Fanuc KAREL source: compact_preamble.KL

PROGRAM KD00043
%NOLOCKGROUP
VAR
I:INTEGER;J:INTEGER;B:BOOLEAN;R:REAL;S : STRING[80]
-- UNRESOLVED DECLARATIONS (source type spelling not recovered)
-- C : TYPE_0x0014 (type_u16=0x0014)
BEGIN
I=1
END KD00043
